// TwinCAT 3 PLC project CounterTests
// ProgramVersion: 3.1.4026.22
// libraries:
//   Tc2_Standard, * (Beckhoff Automation GmbH)
//   Tc2_System, * (Beckhoff Automation GmbH)
//   TcUnit, * (www.tcunit.org)
//   B2SignedDelta_Plc,newest,Tc3 Project
// project tree:
//   / PlcTask.TcTTO
//   POUs/ FB_CounterConsumer.TcPOU, MAIN.TcPOU
// real-time tasks:
//   TASK PlcTask: cycle T#10ms, priority 20, ADS port 350

CONFIGURATION CounterTests
    RESOURCE PLC ON TwinCAT3
        TASK PlcTask(INTERVAL := T#10ms, PRIORITY := 20);
        PROGRAM MAIN WITH PlcTask : MAIN;
    END_RESOURCE
END_CONFIGURATION

// ---- POUs/MAIN.TcPOU
PROGRAM MAIN
VAR
END_VAR

END_PROGRAM

// ---- POUs/FB_CounterConsumer.TcPOU
FUNCTION_BLOCK FB_CounterConsumer
VAR
    counter : B2SignedDelta_Plc.FB_Counter;
    delta : DINT;
END_VAR

delta := UDINT_TO_DINT(counter.GetSignedDelta(a := 5, b := 7));

END_FUNCTION_BLOCK
